TYPE "PositioningMachine_Alr"
VERSION : 0.1
// Block: PositioningMachine_Alr
   STRUCT
      AxisNotInOperation : Bool;
      BrakeTimeOut : Bool;
      AxisTorqueLim : Struct
         Error : Bool;
         ErrorId : Word;
      END_STRUCT;
      Ax : TAx_Alarms;
      Fan_M : MotorAlr;
   END_STRUCT;

END_TYPE
